// TIA Portal V16 export
// export: Created 2023-10-30T22:43:50.8953142Z, ExportSetting WithDefaults, DisplayName Totally Integrated Automation Portal, DisplayVersion V16, DisplayName TIA Portal Version Control Interface, DisplayVersion V16, DisplayName TIA Portal Openness, DisplayVersion V16, DisplayName SINAMICS Startdrive Advanced, DisplayVersion V16, DisplayName SINAMICS Startdrive G130, G150, S120, S150, SINAMICS MV, S210, DisplayVersion V16, DisplayName SINAMICS Startdrive G110M, G120, G120C, G120D, G120P, DisplayVersion V16, DisplayName STEP 7 Professional, DisplayVersion V16, DisplayName STEP 7 Safety, DisplayVersion V16, DisplayName WinCC Professional, DisplayVersion V16
DATA_BLOCK "DataLogWrite_DB"   // DB4
// stored: AutoNumber true, DBAccessibleFromOPCUA true, InstanceOfName DataLogWrite_SFB, OfSystemLibElement DataLogWrite, OfSystemLibVersion 1.0
"DataLogWrite_SFB"
   // VAR_INPUT
   //    REQ : Bool;
   // END_VAR
   // VAR_OUTPUT
   //    DONE : Bool;
   //    BUSY : Bool;
   //    ERROR : Bool;
   //    STATUS : Word;
   // END_VAR
   // VAR_IN_OUT
   //    ID : DWord;
   // END_VAR
BEGIN
END_DATA_BLOCK
